	DATA_BLOCK DB124
	TITLE =DBG024G  GERNERAL ELEMENTS +C19
	//COPYRIGHT:    (C) 2009  BUHLER AG, CH-9240 UZWIL, SWITZERLAND
	//
	//PRODUCT:      WinCoS_BIW01_09
	//
	//TITLE:        GERNERAL ELEMENTS +C19
	//                General group DB
	//                Allgemeine Gruppen-DB
	//
	//-------------------------------------------------------------------------
	//
	//IDENT:        AUTHOR:             DEPT:             DATE:
	//
	//P01_DB124.1.0 K.Renz              CSB41             06.Apr.2010
	//              1st Release
	//
	//-------------------------------------------------------------------------
	//
	//PURPOSE:
	//
	//MANUAL :
	//
	//RESTRICTIONS:
	//
	//-------------------------------------------------------------------------
	AUTHOR  : KR
	FAMILY  : USW
	NAME    : DBG024G
	VERSION : 00.00

	FB124
	BEGIN
	      #Gr.Par.ParObjectNo 	:=2400;
	      #Gr.Par.ParIdling      	:=0;
	      #Gr.Par.ParMgr	        :=False;
	      #Gr.Par.ParWgr	        :=False;
	      #Gr.Par.ParGgr	        :=True;
	      #Gr.Par.ParEmptyingTime 	:=0;
	      #Gr.Par.ParHornCode       :=98;
	//Parameter =A-1999-SHE01 : EMERGENCY-OFF CONVEYOR GREEN MALT
	      #A_1999_SHE01.Par.ParObjectNo                             :=2401;
	      #A_1999_SHE01.Par.ParMsgType                              :=7171;
	      #A_1999_SHE01.Par.ParHornCode                             :=2;
	      #A_1999_SHE01.Par.ParDelayChange                          :=0;
	      #A_1999_SHE01.Par.ParDelayTrue                            :=10;
	      #A_1999_SHE01.Par.ParDelayFalse                           :=0;
	      #A_1999_SHE01.Par.ParTimeoutTrue                          :=0;
	      #A_1999_SHE01.Par.ParTimeoutFalse                         :=0;
	      #A_1999_SHE01.Par.ParLogOff                               :=False;
	      #A_1999_SHE01.Par.Par2WorkingCond                         :=False;
	      #A_1999_SHE01.Par.ParFaultRetry                           :=False;
	      #A_1999_SHE01.Par.ParBinLevel                             :=False;
	//
	//
	//Parameter =A-1999-SHE02 : EMERGENCY-OFF CONVEYOR GREEN MALT
	      #A_1999_SHE02.Par.ParObjectNo                             :=2402;
	      #A_1999_SHE02.Par.ParMsgType                              :=7171;
	      #A_1999_SHE02.Par.ParHornCode                             :=2;
	      #A_1999_SHE02.Par.ParDelayChange                          :=0;
	      #A_1999_SHE02.Par.ParDelayTrue                            :=10;
	      #A_1999_SHE02.Par.ParDelayFalse                           :=0;
	      #A_1999_SHE02.Par.ParTimeoutTrue                          :=0;
	      #A_1999_SHE02.Par.ParTimeoutFalse                         :=0;
	      #A_1999_SHE02.Par.ParLogOff                               :=False;
	      #A_1999_SHE02.Par.Par2WorkingCond                         :=False;
	      #A_1999_SHE02.Par.ParFaultRetry                           :=False;
	      #A_1999_SHE02.Par.ParBinLevel                             :=False;
	//
	//
	//Parameter =A-19-A040Z1 : POWER SUPPLY FAILURE +C19
	      #A_19_A040Z1.Par.ParObjectNo                             :=2403;
	      #A_19_A040Z1.Par.ParMsgType                              :=7135;
	      #A_19_A040Z1.Par.ParHornCode                             :=2;
	      #A_19_A040Z1.Par.ParDelayChange                          :=0;
	      #A_19_A040Z1.Par.ParDelayTrue                            :=10;
	      #A_19_A040Z1.Par.ParDelayFalse                           :=0;
	      #A_19_A040Z1.Par.ParTimeoutTrue                          :=0;
	      #A_19_A040Z1.Par.ParTimeoutFalse                         :=0;
	      #A_19_A040Z1.Par.ParLogOff                               :=False;
	      #A_19_A040Z1.Par.Par2WorkingCond                         :=False;
	      #A_19_A040Z1.Par.ParFaultRetry                           :=False;
	      #A_19_A040Z1.Par.ParBinLevel                             :=False;
	//
	//
	//Parameter =A-19-A097Z1 : EMERGENCY-STOP +C19
	      #A_19_A097Z1.Par.ParObjectNo                             :=2404;
	      #A_19_A097Z1.Par.ParMsgType                              :=7171;
	      #A_19_A097Z1.Par.ParHornCode                             :=2;
	      #A_19_A097Z1.Par.ParDelayChange                          :=0;
	      #A_19_A097Z1.Par.ParDelayTrue                            :=10;
	      #A_19_A097Z1.Par.ParDelayFalse                           :=0;
	      #A_19_A097Z1.Par.ParTimeoutTrue                          :=0;
	      #A_19_A097Z1.Par.ParTimeoutFalse                         :=0;
	      #A_19_A097Z1.Par.ParLogOff                               :=False;
	      #A_19_A097Z1.Par.Par2WorkingCond                         :=False;
	      #A_19_A097Z1.Par.ParFaultRetry                           :=False;
	      #A_19_A097Z1.Par.ParBinLevel                             :=False;
	//
	//
	//Parameter =A-19-K091Z1 : FUSE SWITCH OFF +C19
	      #A_19_K091Z1.Par.ParObjectNo                             :=2405;
	      #A_19_K091Z1.Par.ParMsgType                              :=7135;
	      #A_19_K091Z1.Par.ParHornCode                             :=2;
	      #A_19_K091Z1.Par.ParDelayChange                          :=0;
	      #A_19_K091Z1.Par.ParDelayTrue                            :=10;
	      #A_19_K091Z1.Par.ParDelayFalse                           :=0;
	      #A_19_K091Z1.Par.ParTimeoutTrue                          :=0;
	      #A_19_K091Z1.Par.ParTimeoutFalse                         :=0;
	      #A_19_K091Z1.Par.ParLogOff                               :=False;
	      #A_19_K091Z1.Par.Par2WorkingCond                         :=False;
	      #A_19_K091Z1.Par.ParFaultRetry                           :=False;
	      #A_19_K091Z1.Par.ParBinLevel                             :=False;
	//
	//
	//Parameter =A-19-S/H097Z1 : OPERATING ON +C19
	      #A_19_S_H097Z1.Par.ParObjectNo                             :=2406;
	      #A_19_S_H097Z1.Par.ParMsgType                              :=7154;
	      #A_19_S_H097Z1.Par.ParHornCode                             :=2;
	      #A_19_S_H097Z1.Par.ParDelayChange                          :=0;
	      #A_19_S_H097Z1.Par.ParDelayTrue                            :=10;
	      #A_19_S_H097Z1.Par.ParDelayFalse                           :=0;
	      #A_19_S_H097Z1.Par.ParTimeoutTrue                          :=0;
	      #A_19_S_H097Z1.Par.ParTimeoutFalse                         :=0;
	      #A_19_S_H097Z1.Par.ParLogOff                               :=False;
	      #A_19_S_H097Z1.Par.Par2WorkingCond                         :=False;
	      #A_19_S_H097Z1.Par.ParFaultRetry                           :=False;
	      #A_19_S_H097Z1.Par.ParBinLevel                             :=False;
	//
	//
	END_DATA_BLOCK
